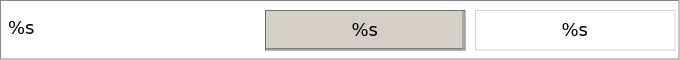
VISUALIZATION SingleRecipesParameterTypeBool_1  // 680x60
VAR_IN_OUT
	stRecipeParameter : ST_VisuCtrlRecipeParameter;
END_VAR
    Textfield (475,10 200x40), "%s", text variable: stRecipeParameter.sFileValue
    Textfield (5,8 250x40), "%s", text variable: stRecipeParameter.sName
    Button (265,10 200x40), "%s", text variable: stRecipeParameter.sName
        toggle stRecipeParameter.bValue
END_VISUALIZATION

(* stored: Version 1.1.0.1, ProductVersion 3.1.4024.12
   Visu SingleRecipesParameterTypeBool_1: Id {659bc801-6340-4889-bc02-c116660d1ff5} *)
